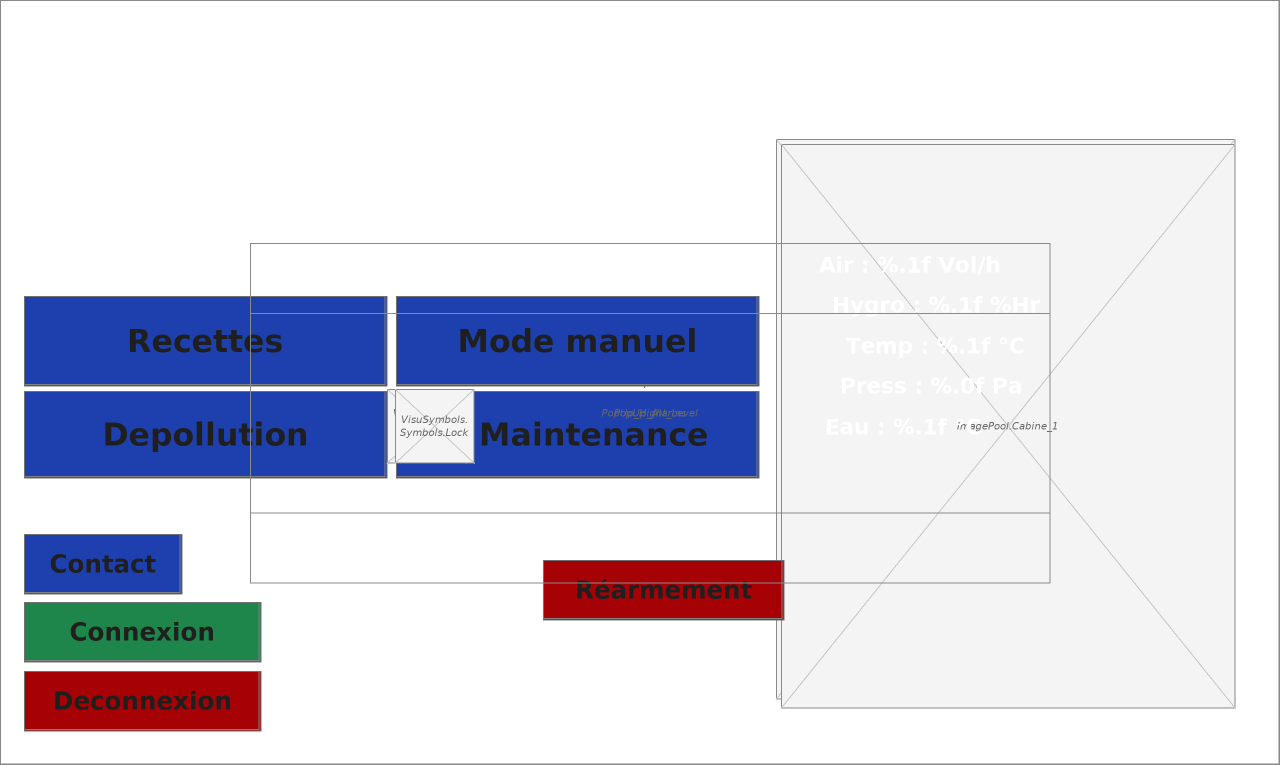
VISUALIZATION menu  // 1280x765
    Frame (0,0 1280x765)
        shows masque()
    Image (776,139 459x560), image: ImagePool.Cabine-2
    Polygon (802,613) (940,653) (1079,687) (1152,653) (1225,613), colour variable: GVL_Visu.Couleur_Cabine
    Polygon (804,613) (802,215) (1081,156) (1222,222) (1223,613), colour variable: GVL_Visu.Couleur_Cabine
    Button (24,391 363x87), "Depollution"
        OnMouseDown: change screen: Depollution
    Button (24,602 237x60), "Connexion"
        OnMouseDown: VisuUserMgmt Type=Login
    Button (24,296 363x90), "Recettes"
        OnMouseDown: change screen: Sel_Recettes
    Image (781,144 454x564), image: ImagePool.Cabine_1
        OnMouseDown: OpenDialog Dialog=Actionneurs, OpenModal=True, OpenCentered=True
    Group (387,389 372x89)
        Button (9,2 363x87), "Maintenance"
            OnMouseDown: execute {
                IF (Option_RegSouf_Ultrason OR Option_Reg_Etanche_Ext OR Option_V3V_EauMitig)
                	THEN
                	VisuElems.CURRENTVISU := 'Maintenance_1';
                	ELSIF (Option_Douche OR Option_Lavabo)
                		THEN
                		VisuElems.CURRENTVISU := 'Maintenance_2';
                	ELSIF (Option_Bas_Debit OR Option_Douchette OR Option_NEP)
                		THEN
                		VisuElems.CURRENTVISU := 'Maintenance_3';
                	ELSIF (Option_WC_GV OR Option_WC_PV OR Option_Prise)
                		THEN
                		VisuElems.CURRENTVISU := 'Maintenance_4';
                	ELSIF (Option_Cabine_Climatique)
                		THEN
                		VisuElems.CURRENTVISU := 'Maintenance_5';
                	ELSE
                	VisuElems.CURRENTVISU := 'Maintenance_6';
                END_IF
            }
        Image (0,0 79x74), invisible if: NOT GVL_Visu.Etat_Connexion, image: VisuSymbols.Symbols.LockOpen
        Image (8,0 79x74), invisible if: GVL_Visu.Etat_Connexion, image: VisuSymbols.Symbols.Lock
    Button (24,671 237x60), "Deconnexion"
        OnMouseDown: VisuUserMgmt Type=Logout
    Button (24,534 158x60), "Contact"
        OnMouseDown: change screen: Accueil
    Button (543,560 241x60), "Réarmement", invisible if: NOT Condi_Affich_Rearm
        OnMouseDown: toggle Cmd_Rearmement
    Group (816,245 317x202)
        Rectangle (6,162 290x40), "Eau : %.1f °C", text variable: MES_Temp_Eau_Mitige_General
        Rectangle (13,40 290x40), "Hygro : %.1f %Hr", text variable: Tab_MES_Sonde_Hygro_Amb.R_MesCor
        Rectangle (27,81 290x40), "Temp : %.1f °C", text variable: Tab_MES_Sonde_Temp_Amb.R_MesCor
        Rectangle (0,0 290x40), "Air : %.1f Vol/h", text variable: MES_Debit_Volh_Soufflage, invisible if: TRUE
        Rectangle (21,121 290x40), "Press : %.0f Pa", text variable: Tab_MES_Sonde_Press_Cab.R_MesCor
    Button (396,296 363x90), "Mode manuel"
        OnMouseDown: change screen: ModeManuel
    Group (250,243 800x340)
        Frame (0,0 800x340), invisible if: NOT GVL_Visu.Affichage_PopUp_Alarm
            shows PopUp_Alarms()
        Frame (0,70 800x200), invisible if: NOT GVL_Visu.Affichage_PopUp_HightLevel
            shows PopUp_Hight_Level()
END_VISUALIZATION

(* stored: Version 1.1.0.1, ProductVersion 3.1.4024.16
   Visu menu: Id {a3cf5cc2-181a-488f-ac8a-3c275bd43792} *)
